INTERFACE PUBLIC StoppedCommands EXTENDS ClearedStateCommands, ResettableStateCommands

END_INTERFACE

(* stored: Version 1.1.0.1, ProductVersion 3.1.4026.18
   Itf StoppedCommands: Id {1719d416-8cac-0ada-1b61-0b25b7a48bba} *)
